Staubli VAL3: writeCNV.pgx

program writeCNV(num& x_nError[] (dimensions=1))
  local bool l_bQuit
  local bool l_bResult
  local num l_nError
  local num l_nStep
  local num l_nValue
  local string l_sErrorMsg
  local string l_sSubString
  local string l_sValue
begin
  // This program initializes the parameters of the conveyor library
  // according to the values of the conveyor page in the settings menu
  // of the wizard.
  //
  //----------------------------------------------------------------
  x_nError=0
  l_nStep=0
  // Update variables of the conveyor library
  resize(sCaption,1,pg:nNumOfTxtBox)
  call pg:getCaption(sCaption)
  //
  l_bQuit=false
  do
    switch l_nStep
      //*** FIELD ENCODER LIBRARY
      case 0
        // Name of the encoder library
        call pg:getFieldValue(sCaption[0],l_sValue,l_nError)
        // checks if encoder library is loadable
        l_nError=enc:libLoad(cfg:sPATHENCODER+l_sValue)
        if l_nError==0
          cnv:sEncoderLib=l_sValue
          l_nStep=10
        else
          x_nError=31
          l_sSubString=cfg:sPATHENCODER+l_sValue
          call ut:addStrToString(lang:sListOfMessage[x_nError],l_sErrorMsg,"",l_sSubString)
          call ut:addNumToString(l_sErrorMsg,l_sErrorMsg,"",l_nError)
          popUpMsg(l_sErrorMsg)
          l_bQuit=true
        endIf
      break
      //*** FIELD DETECTION LIBRARY
      case 10
        // Name of the detection library
        call pg:getFieldValue(sCaption[1],l_sValue,l_nError)
        // checks if detection library is loadable
        l_nError=det:libLoad(cfg:sPATHDETECTION+l_sValue)
        if l_nError==0
          cnv:sDetectionLib=l_sValue
          l_nStep=20
        else
          x_nError=32
          l_sSubString=cfg:sPATHENCODER+l_sValue
          call ut:addStrToString(lang:sListOfMessage[x_nError],l_sErrorMsg,"",l_sSubString)
          call ut:addNumToString(l_sErrorMsg,l_sErrorMsg,"",l_nError)
          popUpMsg(l_sErrorMsg)
          l_bQuit=true
        endIf
      break
      //*** FIELD ThruUpLim
      case 20
        call pg:getFieldValue(sCaption[5],l_sValue,l_nError)
        if l_sValue!=lang:sNONE
          if out:libExist(l_sValue)
            cnv:sUpLimSigName=l_sValue
          else
            x_nError=27
            l_sErrorMsg=lang:sListOfMessage[x_nError]
            popUpMsg(l_sErrorMsg)
            l_bQuit=true
          endIf
        else
          cnv:sUpLimSigName=lang:sNONE
        endIf
        l_nStep=30
      break
      //*** FIELD ThruDwnLim
      case 30
        call pg:getFieldValue(sCaption[6],l_sValue,l_nError)
        if l_sValue!=lang:sNONE
          if out:libExist(l_sValue)
            cnv:sDwnLimSigName=l_sValue
          else
            x_nError=28
            l_sErrorMsg=lang:sListOfMessage[x_nError]
            popUpMsg(l_sErrorMsg)
            l_bQuit=true
          endIf
        else
          cnv:sDwnLimSigName=lang:sNONE
        endIf
        l_nStep=40
      break
      //*** FIELD Event logging
      case 40
        call pg:getFieldValue(sCaption[11],l_sValue,l_nError)
        if l_sValue=="TRUE"
          cnv:bLOG=true
        else
          cnv:bLOG=false
        endIf
        l_nStep=50
      break
      //
      case 50
        // height of the tracking window
        call pg:getFieldValue(sCaption[4],l_sValue,l_nError)
        toNum(l_sValue,cnv:nTrackWinHeight,l_bResult)
        // Buffersize
        call pg:getFieldValue(sCaption[2],l_sValue,l_nError)
        toNum(l_sValue,cnv:nBufferSize,l_bResult)
        // Scale factor
        call pg:getFieldValue(sCaption[3],l_sValue,l_nError)
        toNum(l_sValue,cnv:nENCSCALEFACTOR,l_bResult)
        // Matching tolerance
        call pg:getFieldValue(sCaption[7],l_sValue,l_nError)
        toNum(l_sValue,cnv:nPosMatchTol,l_bResult)
        //  Clock Signal
        call pg:getFieldValue(sCaption[8],l_sValue,l_nError)
        // If an IO name is set for ClockSignal,Check if is a digital IO
        if l_sValue!=lang:sNONE
          getData("out:"+l_sValue,doClock)
          if ioStatus(doClock)>=0
            cnv:sClockSigName=l_sValue
          else
            x_nError=26
            l_sErrorMsg=lang:sListOfMessage[x_nError]
            popUpMsg(l_sErrorMsg)
          endIf
        else
          cnv:sClockSigName=lang:sNONE
        endIf
        //
        // Clock Period
        call pg:getFieldValue(sCaption[9],l_sValue,l_nError)
        toNum(l_sValue,cnv:nClockPeriod,l_bResult)
        // latch lock distance
        call pg:getFieldValue(sCaption[10],l_sValue,l_nError)
        toNum(l_sValue,cnv:nLatchLockDist,l_bResult)
        l_bQuit=true
      break
    endSwitch
  until (l_bQuit==true)
end
